TYPE T_JCL_ID :
STRUCT
	Jcl: INT;
	Jcl_Tcp: INT;
END_STRUCT
END_TYPE

(* stored: Version 1.1.0.1, ProductVersion 3.1.0.26
   DUT T_JCL_ID: Id {aeaf3c7e-c16f-46ae-80f4-c612369ad99f} *)
